PROGRAM Blinker
VAR
	
	fbBlinker1								:FB_Blinker;
	tTurnOffDelayB1							:TIME := T#1S;
	fbBlinker2								:FB_Blinker;
	
END_VAR
(* End *)

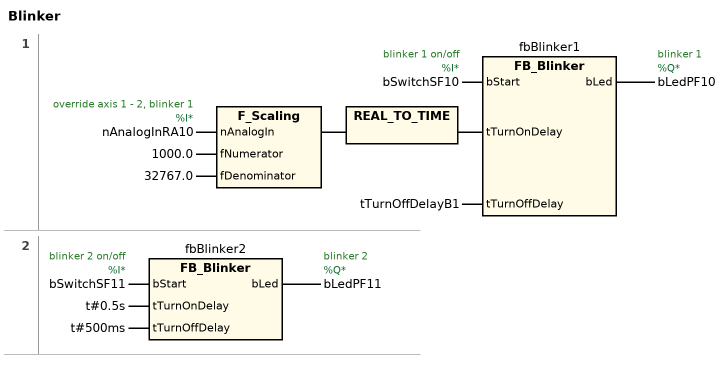
// NETWORK 1
//   bSwitchSF10: blinker 1 on/off | AT %I*
//   nAnalogInRA10: override axis 1 - 2, blinker 1 | AT %I*
//   bLedPF10: blinker 1 | AT %Q*
fbBlinker1(
    bStart := bSwitchSF10,
    tTurnOnDelay := REAL_TO_TIME(F_Scaling(nAnalogIn := nAnalogInRA10, fNumerator := 1000.0, fDenominator := 32767.0)),
    tTurnOffDelay := tTurnOffDelayB1); // FB_Blinker
bLedPF10 := fbBlinker1.bLed;

// NETWORK 2
//   bSwitchSF11: blinker 2 on/off | AT %I*
//   bLedPF11: blinker 2 | AT %Q*
fbBlinker2(bStart := bSwitchSF11, tTurnOnDelay := t#0.5s, tTurnOffDelay := t#500ms); // FB_Blinker
bLedPF11 := fbBlinker2.bLed;

END_PROGRAM

(* stored: Version 1.1.0.1
   POU Blinker: Id {412a77ed-f576-470f-97fb-b89f207e2796}, SpecialFunc None *)
